{attribute 'qualified_only'}
{attribute 'strict'}
TYPE TrackState :
(
	WAIT_FOR_COMMAND	:= 0,
	SETUP_FUNCTION		:= 100,
	MONITOR_RESPONSE	:= 110,
	REQUIRED_DELAY		:= 200,
	CLEAN_UP			:= 300,
	WAIT_END			:= 1000,
	ERROR				:= 9000
);
END_TYPE

(* stored: Version 1.1.0.1, ProductVersion 3.1.4026.8
   DUT TrackState: Id {b8cf507c-0268-0834-24f4-900859769bcf} *)
